FUNCTION ifExprFunc5: DINT
VAR_INPUT
    state: STATE;
END_VAR


        IF (state.dvar_M_p_vt) THEN
    ifExprFunc5 := 8;
ELSIF (state.dvar_M_p_vf) THEN
    ifExprFunc5 := 9;
ELSE
    ifExprFunc5 := 10;
END_IF;

END_FUNCTION

(* stored: ProductVersion 3.1.0.18, Version 1.1.0.1 *)
